// Mitsubishi GX Works2 project: programme luxia plc final   PLC: FX3U/FX3UC

PROGRAM MAIN
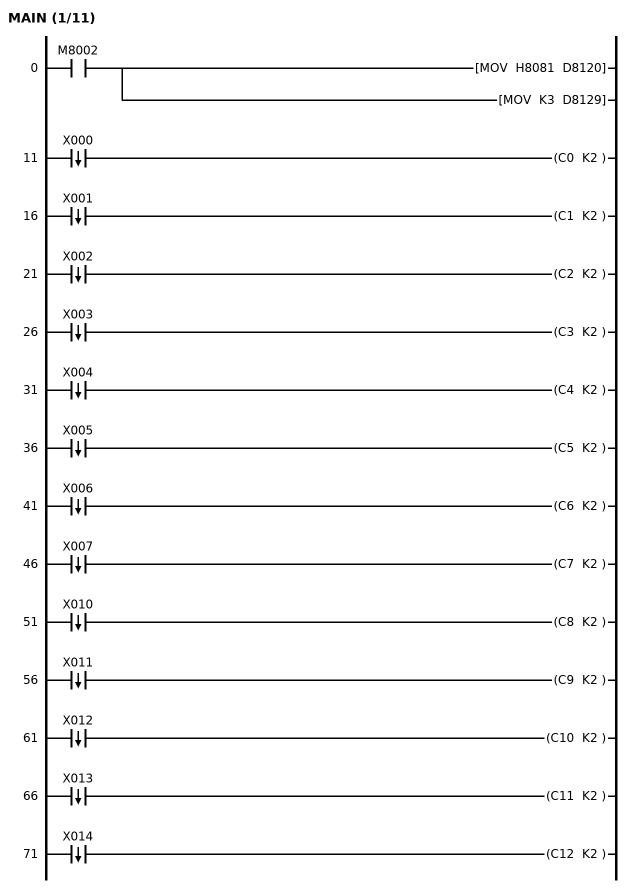
0     LD      M8002
      MOV     H8081 D8120
      MOV     K3 D8129
11    LDF     X000
      OUT     C0 K2
16    LDF     X001
      OUT     C1 K2
21    LDF     X002
      OUT     C2 K2
26    LDF     X003
      OUT     C3 K2
31    LDF     X004
      OUT     C4 K2
36    LDF     X005
      OUT     C5 K2
41    LDF     X006
      OUT     C6 K2
46    LDF     X007
      OUT     C7 K2
51    LDF     X010
      OUT     C8 K2
56    LDF     X011
      OUT     C9 K2
61    LDF     X012
      OUT     C10 K2
66    LDF     X013
      OUT     C11 K2
71    LDF     X014
      OUT     C12 K2
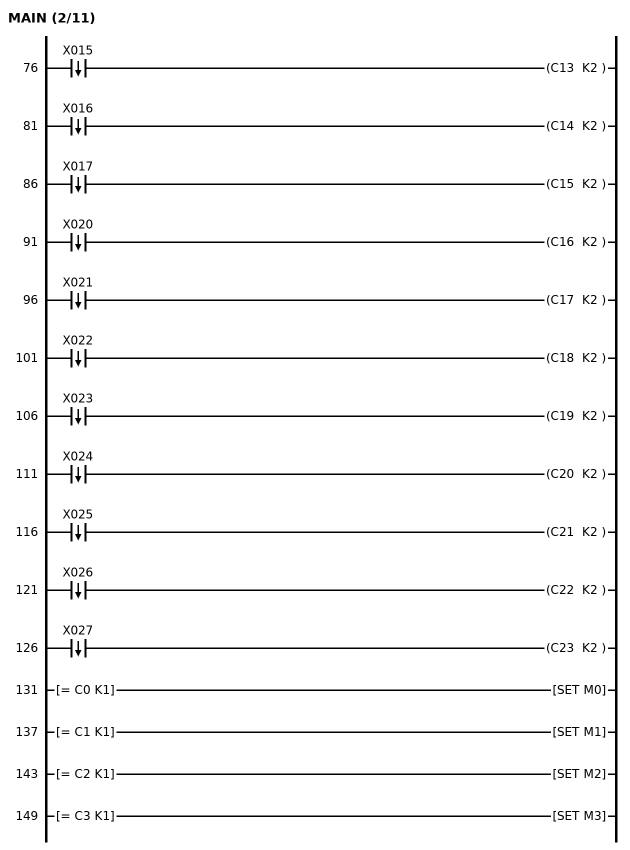
76    LDF     X015
      OUT     C13 K2
81    LDF     X016
      OUT     C14 K2
86    LDF     X017
      OUT     C15 K2
91    LDF     X020
      OUT     C16 K2
96    LDF     X021
      OUT     C17 K2
101   LDF     X022
      OUT     C18 K2
106   LDF     X023
      OUT     C19 K2
111   LDF     X024
      OUT     C20 K2
116   LDF     X025
      OUT     C21 K2
121   LDF     X026
      OUT     C22 K2
126   LDF     X027
      OUT     C23 K2
131   LD=     C0 K1
      SET     M0
137   LD=     C1 K1
      SET     M1
143   LD=     C2 K1
      SET     M2
149   LD=     C3 K1
      SET     M3
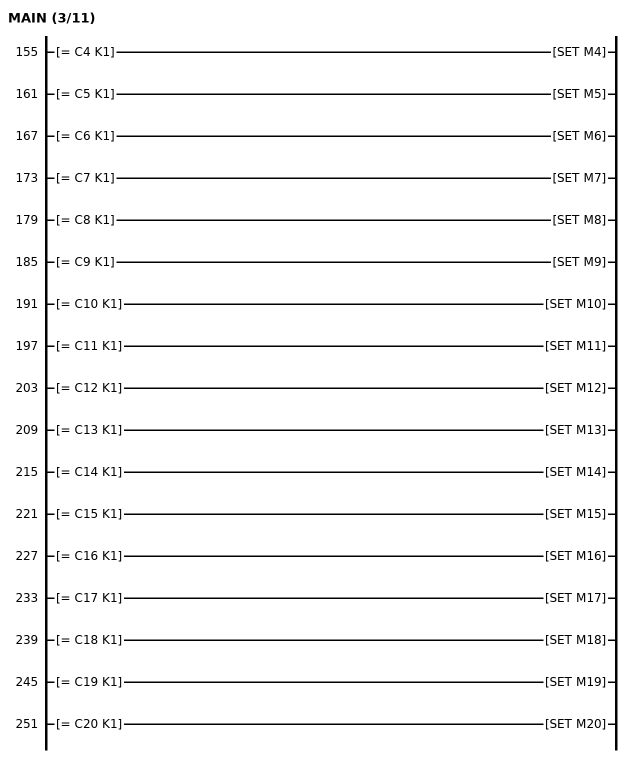
155   LD=     C4 K1
      SET     M4
161   LD=     C5 K1
      SET     M5
167   LD=     C6 K1
      SET     M6
173   LD=     C7 K1
      SET     M7
179   LD=     C8 K1
      SET     M8
185   LD=     C9 K1
      SET     M9
191   LD=     C10 K1
      SET     M10
197   LD=     C11 K1
      SET     M11
203   LD=     C12 K1
      SET     M12
209   LD=     C13 K1
      SET     M13
215   LD=     C14 K1
      SET     M14
221   LD=     C15 K1
      SET     M15
227   LD=     C16 K1
      SET     M16
233   LD=     C17 K1
      SET     M17
239   LD=     C18 K1
      SET     M18
245   LD=     C19 K1
      SET     M19
251   LD=     C20 K1
      SET     M20
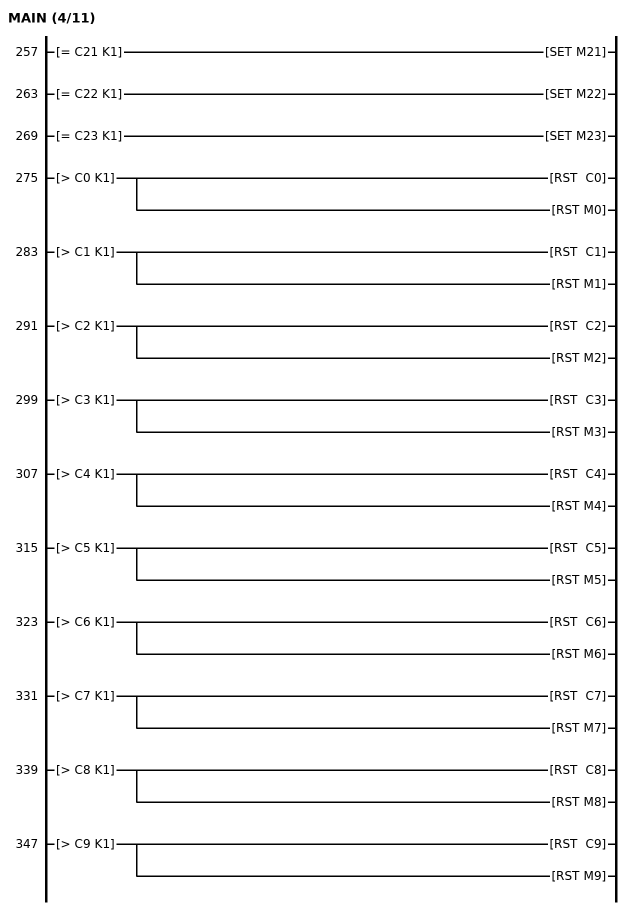
257   LD=     C21 K1
      SET     M21
263   LD=     C22 K1
      SET     M22
269   LD=     C23 K1
      SET     M23
275   LD>     C0 K1
      RST     C0
      RST     M0
283   LD>     C1 K1
      RST     C1
      RST     M1
291   LD>     C2 K1
      RST     C2
      RST     M2
299   LD>     C3 K1
      RST     C3
      RST     M3
307   LD>     C4 K1
      RST     C4
      RST     M4
315   LD>     C5 K1
      RST     C5
      RST     M5
323   LD>     C6 K1
      RST     C6
      RST     M6
331   LD>     C7 K1
      RST     C7
      RST     M7
339   LD>     C8 K1
      RST     C8
      RST     M8
347   LD>     C9 K1
      RST     C9
      RST     M9
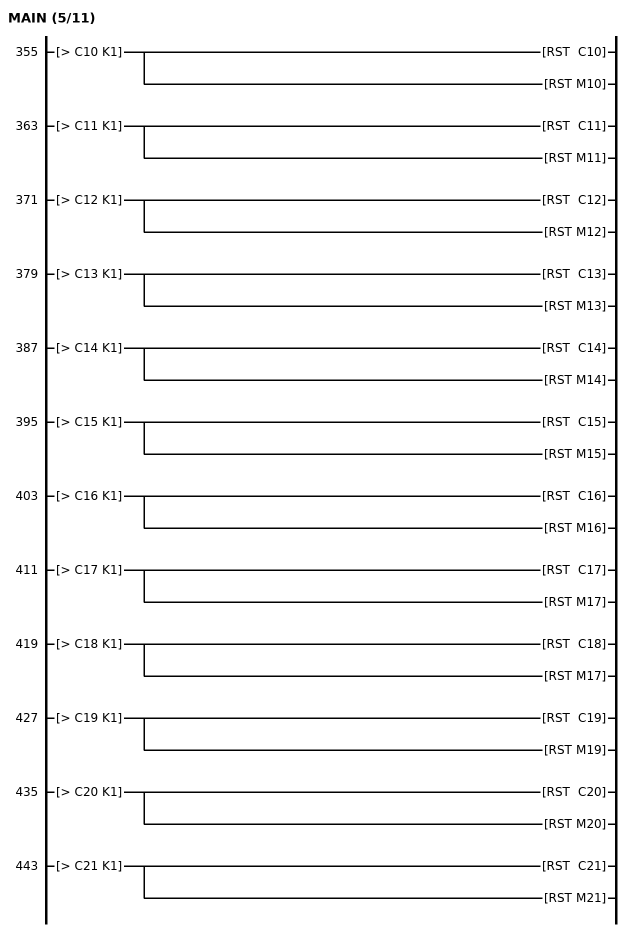
355   LD>     C10 K1
      RST     C10
      RST     M10
363   LD>     C11 K1
      RST     C11
      RST     M11
371   LD>     C12 K1
      RST     C12
      RST     M12
379   LD>     C13 K1
      RST     C13
      RST     M13
387   LD>     C14 K1
      RST     C14
      RST     M14
395   LD>     C15 K1
      RST     C15
      RST     M15
403   LD>     C16 K1
      RST     C16
      RST     M16
411   LD>     C17 K1
      RST     C17
      RST     M17
419   LD>     C18 K1
      RST     C18
      RST     M17
427   LD>     C19 K1
      RST     C19
      RST     M19
435   LD>     C20 K1
      RST     C20
      RST     M20
443   LD>     C21 K1
      RST     C21
      RST     M21
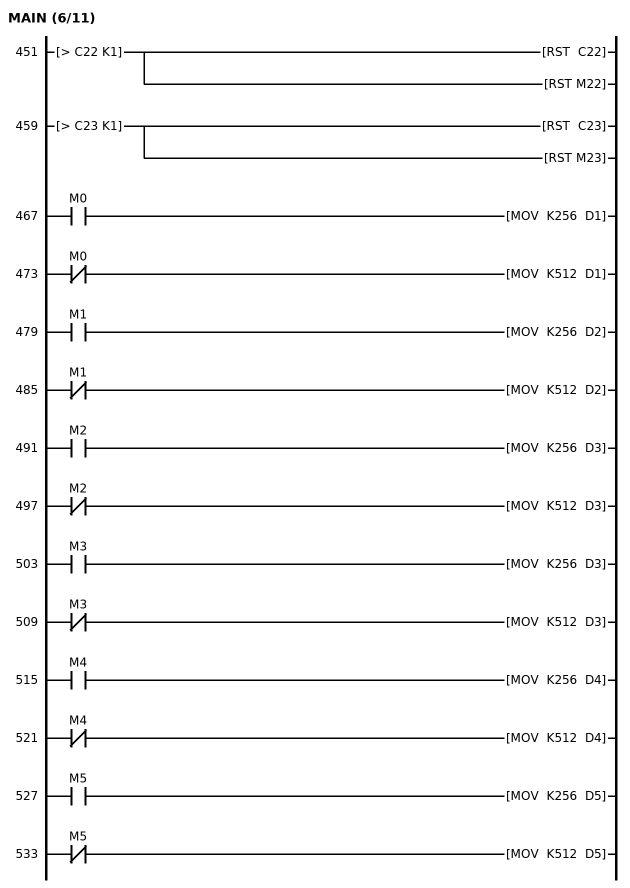
451   LD>     C22 K1
      RST     C22
      RST     M22
459   LD>     C23 K1
      RST     C23
      RST     M23
467   LD      M0
      MOV     K256 D1
473   LDI     M0
      MOV     K512 D1
479   LD      M1
      MOV     K256 D2
485   LDI     M1
      MOV     K512 D2
491   LD      M2
      MOV     K256 D3
497   LDI     M2
      MOV     K512 D3
503   LD      M3
      MOV     K256 D3
509   LDI     M3
      MOV     K512 D3
515   LD      M4
      MOV     K256 D4
521   LDI     M4
      MOV     K512 D4
527   LD      M5
      MOV     K256 D5
533   LDI     M5
      MOV     K512 D5
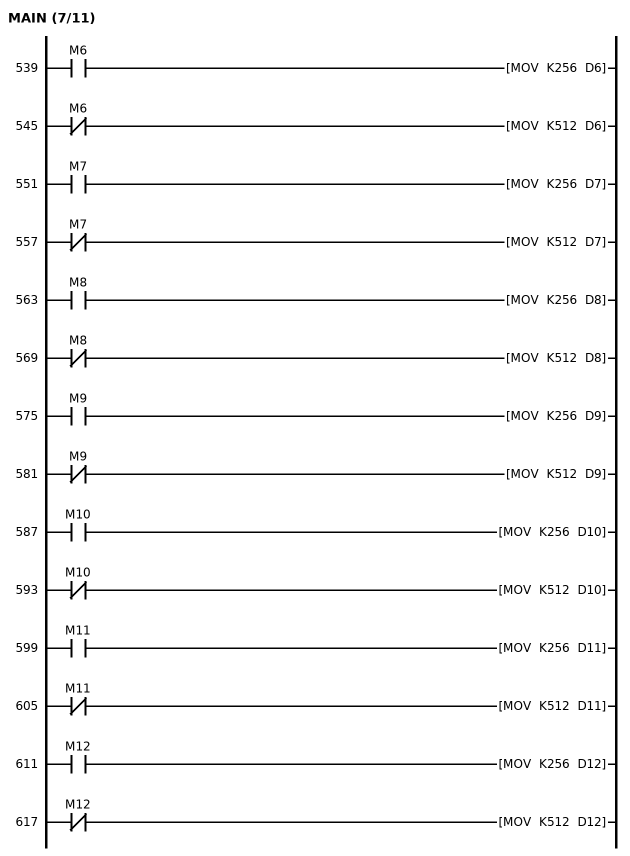
539   LD      M6
      MOV     K256 D6
545   LDI     M6
      MOV     K512 D6
551   LD      M7
      MOV     K256 D7
557   LDI     M7
      MOV     K512 D7
563   LD      M8
      MOV     K256 D8
569   LDI     M8
      MOV     K512 D8
575   LD      M9
      MOV     K256 D9
581   LDI     M9
      MOV     K512 D9
587   LD      M10
      MOV     K256 D10
593   LDI     M10
      MOV     K512 D10
599   LD      M11
      MOV     K256 D11
605   LDI     M11
      MOV     K512 D11
611   LD      M12
      MOV     K256 D12
617   LDI     M12
      MOV     K512 D12
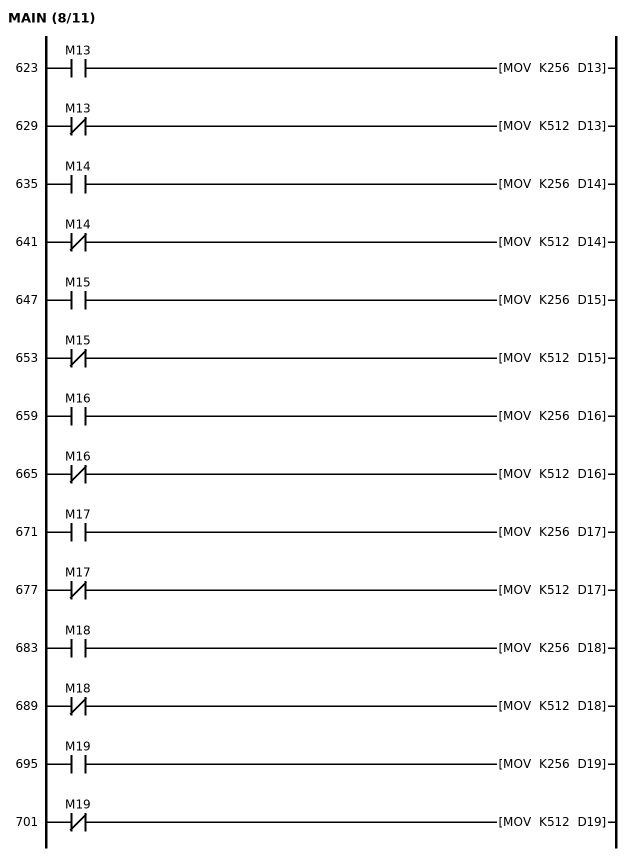
623   LD      M13
      MOV     K256 D13
629   LDI     M13
      MOV     K512 D13
635   LD      M14
      MOV     K256 D14
641   LDI     M14
      MOV     K512 D14
647   LD      M15
      MOV     K256 D15
653   LDI     M15
      MOV     K512 D15
659   LD      M16
      MOV     K256 D16
665   LDI     M16
      MOV     K512 D16
671   LD      M17
      MOV     K256 D17
677   LDI     M17
      MOV     K512 D17
683   LD      M18
      MOV     K256 D18
689   LDI     M18
      MOV     K512 D18
695   LD      M19
      MOV     K256 D19
701   LDI     M19
      MOV     K512 D19
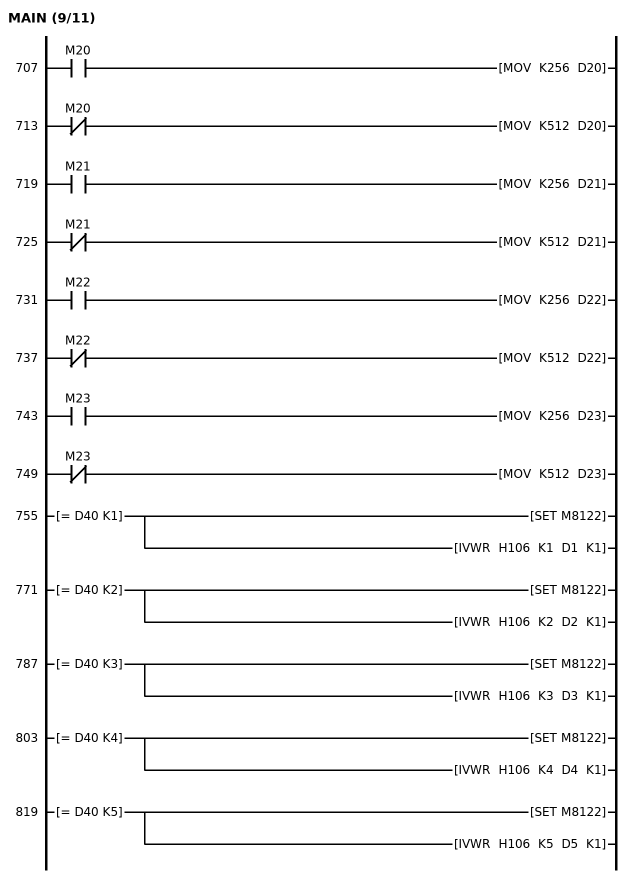
707   LD      M20
      MOV     K256 D20
713   LDI     M20
      MOV     K512 D20
719   LD      M21
      MOV     K256 D21
725   LDI     M21
      MOV     K512 D21
731   LD      M22
      MOV     K256 D22
737   LDI     M22
      MOV     K512 D22
743   LD      M23
      MOV     K256 D23
749   LDI     M23
      MOV     K512 D23
755   LD=     D40 K1
      SET     M8122
      IVWR    H106 K1 D1 K1
771   LD=     D40 K2
      SET     M8122
      IVWR    H106 K2 D2 K1
787   LD=     D40 K3
      SET     M8122
      IVWR    H106 K3 D3 K1
803   LD=     D40 K4
      SET     M8122
      IVWR    H106 K4 D4 K1
819   LD=     D40 K5
      SET     M8122
      IVWR    H106 K5 D5 K1
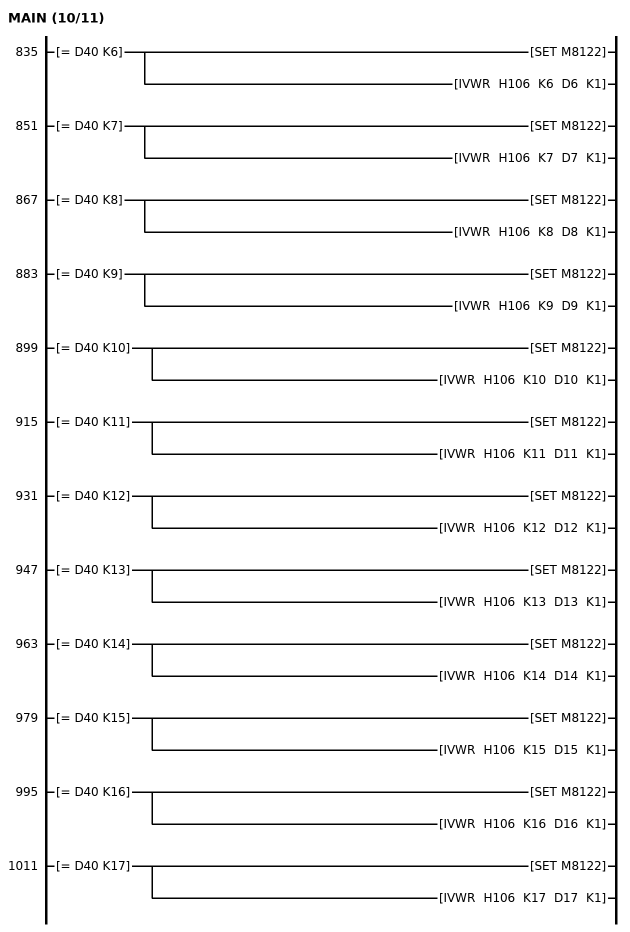
835   LD=     D40 K6
      SET     M8122
      IVWR    H106 K6 D6 K1
851   LD=     D40 K7
      SET     M8122
      IVWR    H106 K7 D7 K1
867   LD=     D40 K8
      SET     M8122
      IVWR    H106 K8 D8 K1
883   LD=     D40 K9
      SET     M8122
      IVWR    H106 K9 D9 K1
899   LD=     D40 K10
      SET     M8122
      IVWR    H106 K10 D10 K1
915   LD=     D40 K11
      SET     M8122
      IVWR    H106 K11 D11 K1
931   LD=     D40 K12
      SET     M8122
      IVWR    H106 K12 D12 K1
947   LD=     D40 K13
      SET     M8122
      IVWR    H106 K13 D13 K1
963   LD=     D40 K14
      SET     M8122
      IVWR    H106 K14 D14 K1
979   LD=     D40 K15
      SET     M8122
      IVWR    H106 K15 D15 K1
995   LD=     D40 K16
      SET     M8122
      IVWR    H106 K16 D16 K1
1011  LD=     D40 K17
      SET     M8122
      IVWR    H106 K17 D17 K1
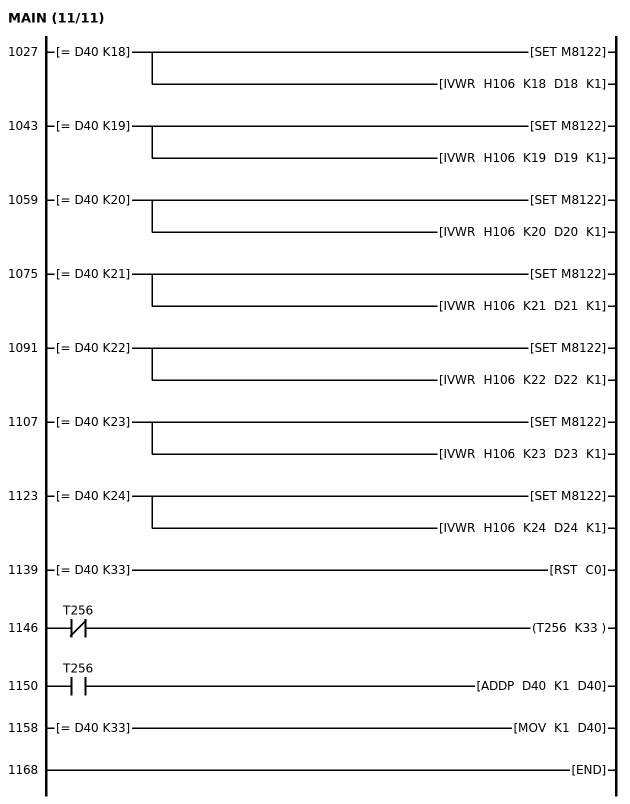
1027  LD=     D40 K18
      SET     M8122
      IVWR    H106 K18 D18 K1
1043  LD=     D40 K19
      SET     M8122
      IVWR    H106 K19 D19 K1
1059  LD=     D40 K20
      SET     M8122
      IVWR    H106 K20 D20 K1
1075  LD=     D40 K21
      SET     M8122
      IVWR    H106 K21 D21 K1
1091  LD=     D40 K22
      SET     M8122
      IVWR    H106 K22 D22 K1
1107  LD=     D40 K23
      SET     M8122
      IVWR    H106 K23 D23 K1
1123  LD=     D40 K24
      SET     M8122
      IVWR    H106 K24 D24 K1
1139  LD=     D40 K33
      RST     C0
1146  LDI     T256
      OUT     T256 K33
1150  LD      T256
      ADDP    D40 K1 D40
1158  LD=     D40 K33
      MOV     K1 D40
1168  END
END_PROGRAM
